FUNCTION_BLOCK Motor
VAR_INPUT
	MotorInputs : MotorInputvariables;
END_VAR
VAR_OUTPUT
	MotorOutputs : MotorOutputVariables;
END_VAR
VAR
	Start : BOOL;
	Stop : BOOL;
END_VAR

Start := MotorInputs.Start;
Stop := MotorInputs.Stop;

IF Start AND Stop = FALSE AND MotorInputs.Oveload = FALSE THEN
	MotorOutputs.Coil := TRUE;
ELSE
	MotorOutputs.Coil := FALSE;
	
END_IF

END_FUNCTION_BLOCK

(* stored: Version 1.1.0.1, ProductVersion 3.1.4024.9
   POU Motor: Id {86737985-3d77-4234-9009-bf8bef62507e}, SpecialFunc None *)
